FUNCTION_BLOCK FB_Estacion
VAR_INPUT
    UnidadesSolicitadas: UINT := 1;
    
	TiempoRetenedor: TIME := T#1S;
	TiempoSeparador: TIME := T#1S;
	TiempoEntradaPale: TIME := T#1S;
    TiempoSalidaPale: TIME := T#1S;
    TiempoTransferenciPale: TIME := T#1S;
    
	TiempoVerificacion: TIME := T#1S;
	TiempoDesplazador: TIME := T#2S;
    TiempoRechazador: TIME := T#1S;
END_VAR
VAR_OUTPUT
    CondicionInicial: BOOL;
    CondicionMarcha: BOOL;
    UnidadesPendientes: UINT;
    
	i_SelectorManual AT %I*: BOOL;
END_VAR
VAR
    MarchaAutorizada: BOOL;
    TareaFinalizada: BOOL;
    
    UnidadCorrecta: BOOL;
    
    // Variables de entrada
    i_PulsadorEmergencia AT %I*: BOOL;
    // i_SelectorManual AT %I*: BOOL;
    i_PulsadorMarcha AT %I*: BOOL;
    i_PulsadorParada AT %I*: BOOL := TRUE; // Normalmente cerrado
    i_EstacionConectada AT %I*: BOOL := TRUE;
    i_PresenciaPale AT %I*: BOOL;
    i_CodigoPaleBit0 AT %I*: BOOL;
    i_CodigoPaleBit1 AT %I*: BOOL;
    
    i_CodigoPaleBit2 AT %I*: BOOL;
    i_DetectorPresion AT %I*: BOOL := TRUE;
    
    i_DescargadorDetras AT %I*: BOOL := TRUE;
    i_DescargadorDelante AT %I*: BOOL;
    i_DescargadorArriba AT %I*: BOOL := TRUE;
    i_DescargadorAbajo AT %I*: BOOL;
    i_VerificadorArriba AT %I*: BOOL := TRUE;
    i_VerificadorAbajo AT %I*: BOOL;
    i_DesplazadorDetras AT %I*: BOOL := TRUE;
    i_EmpujadorDetras AT %I*: BOOL := TRUE;
    
    i_EmpujadorDelante AT %I*: BOOL;
    i_DescargadorVacio AT %I*: BOOL;
    i_PresenciaBase AT %I*: BOOL;
    
    // Variables de salida
    o_DesconectaEstacion AT %Q*: BOOL;
    o_LamparaAlarma AT %Q*: BOOL;
    o_LamparaMarcha AT %Q*: BOOL;
    o_LamparaMaterial AT %Q*: BOOL;
    o_CintaActiva AT %Q*: BOOL;
    o_CintaInvierte AT %Q*: BOOL;
    o_RetenedorBaja AT %Q*: BOOL;
    o_SeparadorSube AT %Q*: BOOL;
    
    o_AvisadorSonoro AT %Q*: BOOL;
    
    o_DescargadorAvanza AT %Q*: BOOL;
    o_DescargadorRetrocede AT %Q*: BOOL;
    o_DescargadorBaja AT %Q*: BOOL;
    o_RechazadorAvanza AT %Q*: BOOL;
    o_VerificardorBaja AT %Q*: BOOL;
    o_DesplazadorAvanza AT %Q*: BOOL;
    o_EmpujadorAvanza AT %Q*: BOOL;
    o_DescargadorSucciona AT %Q*: BOOL;
END_VAR

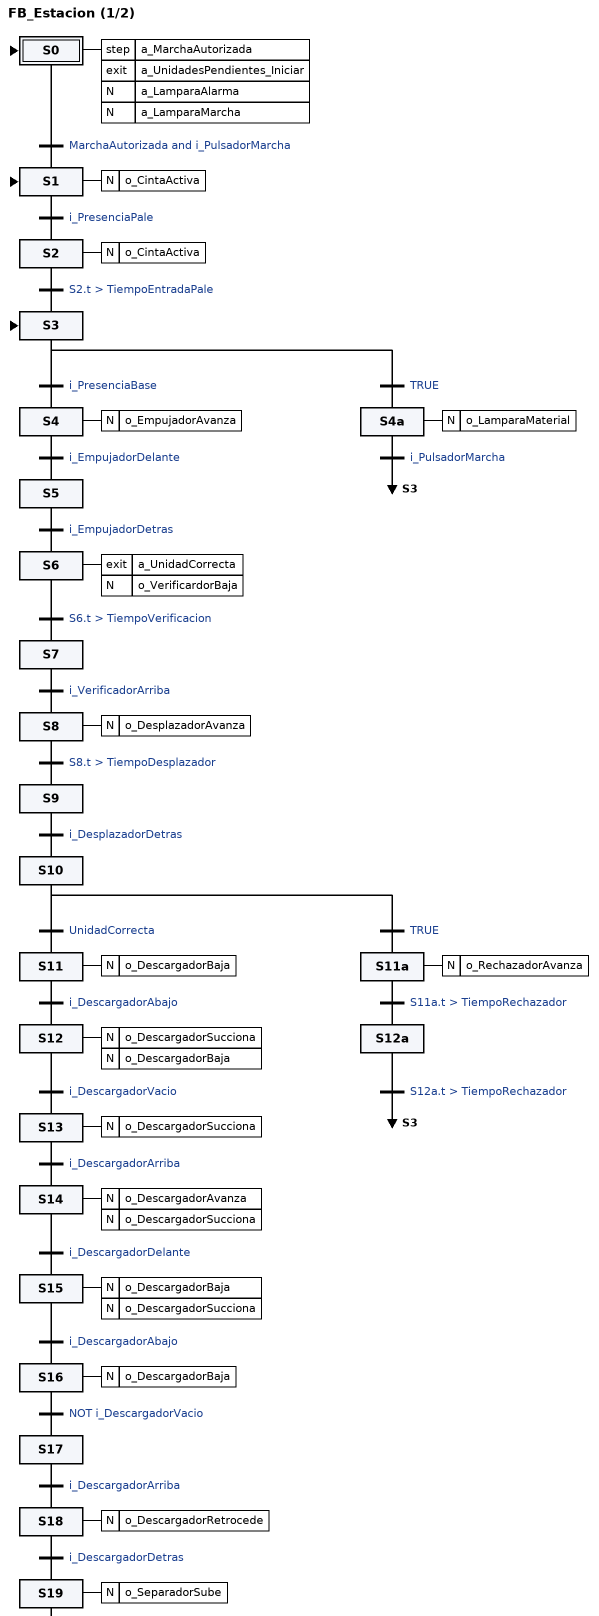
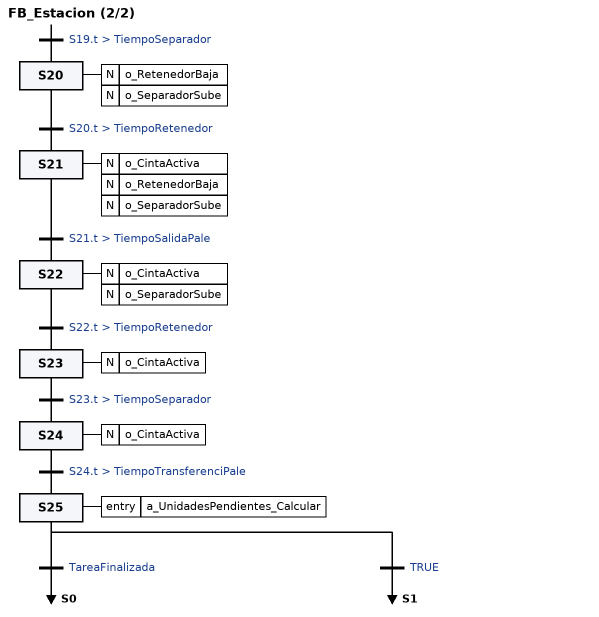
INITIAL_STEP S0:
    a_MarchaAutorizada(N);  // step action
    a_UnidadesPendientes_Iniciar(P0);  // exit action
    a_LamparaAlarma(N);
    a_LamparaMarcha(N);
END_STEP
TRANSITION FROM S0 TO S1
    := MarchaAutorizada and i_PulsadorMarcha;
END_TRANSITION
STEP S1:
    o_CintaActiva(N);
END_STEP
TRANSITION FROM S1 TO S2
    := i_PresenciaPale;
END_TRANSITION
STEP S2:
    o_CintaActiva(N);
END_STEP
TRANSITION FROM S2 TO S3
    := S2.t > TiempoEntradaPale;
END_TRANSITION
STEP S3:
END_STEP
TRANSITION FROM S3 TO S4
    := i_PresenciaBase;
END_TRANSITION
STEP S4:
    o_EmpujadorAvanza(N);
END_STEP
TRANSITION FROM S4 TO S5
    := i_EmpujadorDelante;
END_TRANSITION
STEP S5:
END_STEP
TRANSITION FROM S5 TO S6
    := i_EmpujadorDetras;
END_TRANSITION
STEP S6:
    a_UnidadCorrecta(P0);  // exit action
    o_VerificardorBaja(N);
END_STEP
TRANSITION FROM S6 TO S7
    := S6.t > TiempoVerificacion;
END_TRANSITION
STEP S7:
END_STEP
TRANSITION FROM S7 TO S8
    := i_VerificadorArriba;
END_TRANSITION
STEP S8:
    o_DesplazadorAvanza(N);
END_STEP
TRANSITION FROM S8 TO S9
    := S8.t > TiempoDesplazador;
END_TRANSITION
STEP S9:
END_STEP
TRANSITION FROM S9 TO S10
    := i_DesplazadorDetras;
END_TRANSITION
STEP S10:
END_STEP
TRANSITION FROM S10 TO S11
    := UnidadCorrecta;
END_TRANSITION
STEP S11:
    o_DescargadorBaja(N);
END_STEP
TRANSITION FROM S11 TO S12
    := i_DescargadorAbajo;
END_TRANSITION
STEP S12:
    o_DescargadorSucciona(N);
    o_DescargadorBaja(N);
END_STEP
TRANSITION FROM S12 TO S13
    := i_DescargadorVacio;
END_TRANSITION
STEP S13:
    o_DescargadorSucciona(N);
END_STEP
TRANSITION FROM S13 TO S14
    := i_DescargadorArriba;
END_TRANSITION
STEP S14:
    o_DescargadorAvanza(N);
    o_DescargadorSucciona(N);
END_STEP
TRANSITION FROM S14 TO S15
    := i_DescargadorDelante;
END_TRANSITION
STEP S15:
    o_DescargadorBaja(N);
    o_DescargadorSucciona(N);
END_STEP
TRANSITION FROM S15 TO S16
    := i_DescargadorAbajo;
END_TRANSITION
STEP S16:
    o_DescargadorBaja(N);
END_STEP
TRANSITION FROM S16 TO S17
    := NOT i_DescargadorVacio;
END_TRANSITION
STEP S17:
END_STEP
TRANSITION FROM S17 TO S18
    := i_DescargadorArriba;
END_TRANSITION
STEP S18:
    o_DescargadorRetrocede(N);
END_STEP
TRANSITION FROM S18 TO S19
    := i_DescargadorDetras;
END_TRANSITION
STEP S19:
    o_SeparadorSube(N);
END_STEP
TRANSITION FROM S19 TO S20
    := S19.t > TiempoSeparador;
END_TRANSITION
STEP S20:
    o_RetenedorBaja(N);
    o_SeparadorSube(N);
END_STEP
TRANSITION FROM S20 TO S21
    := S20.t > TiempoRetenedor;
END_TRANSITION
STEP S21:
    o_CintaActiva(N);
    o_RetenedorBaja(N);
    o_SeparadorSube(N);
END_STEP
TRANSITION FROM S21 TO S22
    := S21.t > TiempoSalidaPale;
END_TRANSITION
STEP S22:
    o_CintaActiva(N);
    o_SeparadorSube(N);
END_STEP
TRANSITION FROM S22 TO S23
    := S22.t > TiempoRetenedor;
END_TRANSITION
STEP S23:
    o_CintaActiva(N);
END_STEP
TRANSITION FROM S23 TO S24
    := S23.t > TiempoSeparador;
END_TRANSITION
STEP S24:
    o_CintaActiva(N);
END_STEP
TRANSITION FROM S24 TO S25
    := S24.t > TiempoTransferenciPale;
END_TRANSITION
TRANSITION FROM S10 TO S11a
    := TRUE;
END_TRANSITION
STEP S11a:
    o_RechazadorAvanza(N);
END_STEP
TRANSITION FROM S11a TO S12a
    := S11a.t > TiempoRechazador;
END_TRANSITION
STEP S12a:
END_STEP
TRANSITION FROM S12a TO S3
    := S12a.t > TiempoRechazador;
END_TRANSITION
TRANSITION FROM S3 TO S4a
    := TRUE;
END_TRANSITION
STEP S4a:
    o_LamparaMaterial(N);
END_STEP
TRANSITION FROM S4a TO S3
    := i_PulsadorMarcha;
END_TRANSITION
STEP S25:
    a_UnidadesPendientes_Calcular(P1);  // entry action
END_STEP
TRANSITION FROM S25 TO S0
    := TareaFinalizada;
END_TRANSITION
TRANSITION FROM S25 TO S1
    := TRUE;
END_TRANSITION

ACTION a_CondicionInicial:
CondicionInicial := i_DetectorPresion
    AND i_EstacionConectada
    AND i_EmpujadorDetras
    AND i_VerificadorArriba
    AND i_DesplazadorDetras
    AND i_DescargadorDetras
    AND i_DescargadorArriba;
END_ACTION

ACTION a_LamparaAlarma:
o_LamparaAlarma := (S0.x AND NOT MarchaAutorizada);
END_ACTION

ACTION a_LamparaMarcha:
o_LamparaMarcha := NOT S0.x;
END_ACTION

ACTION a_MarchaAutorizada:
a_CondicionInicial();

CondicionMarcha := (UnidadesSolicitadas > 0);
MarchaAutorizada := CondicionInicial AND CondicionMarcha;
END_ACTION

ACTION a_UnidadCorrecta:
UnidadCorrecta := i_VerificadorAbajo;
END_ACTION

ACTION a_UnidadesPendientes_Calcular:
IF UnidadesPendientes > 0 THEN
    UnidadesPendientes := UnidadesPendientes - 1;
END_IF;

TareaFinalizada := (UnidadesPendientes = 0);
END_ACTION

ACTION a_UnidadesPendientes_Iniciar:
UnidadesPendientes := UnidadesSolicitadas;
END_ACTION

END_FUNCTION_BLOCK

(* stored: Version 1.1.0.1
   POU FB_Estacion: Id {0900b681-9b01-4b7c-9570-85b5f70c48a2}, SpecialFunc None
   Action a_CondicionInicial: Id {da48870b-a9a4-0983-0dbb-cdc36f43067c}
   Action a_LamparaAlarma: Id {cdaafdb1-1d28-0651-0a6c-87941382fa76}
   Action a_LamparaMarcha: Id {4cbaf431-03d8-0f1f-38d2-2bcf9ecda9f9}
   Action a_MarchaAutorizada: Id {50e82557-1c85-084f-13dd-c0ab9e9e78d6}
   Action a_UnidadCorrecta: Id {91682ee4-653b-02b9-0fa3-0ca2fab11185}
   Action a_UnidadesPendientes_Calcular: Id {02a5032b-6e7b-001d-041b-1485fa225e04}
   Action a_UnidadesPendientes_Iniciar: Id {42172e6e-a864-0f61-2d9d-05e86b199c8d} *)
